# EPICS substitutions: db/Festo/ecmcFesto-CMMT-ST.substitutions
file "ecmcFesto-CMM-ST.template" { pattern
  { CH_ID }
  { 01    }
}
